// Mitsubishi GX Works2 project: yudomotmutistep   PLC: Q03UDV

PROGRAM MAIN
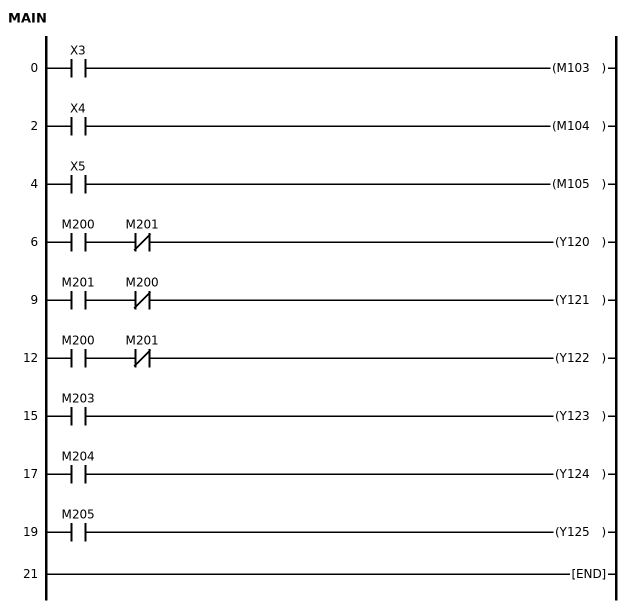
0     LD      X3
      OUT     M103
2     LD      X4
      OUT     M104
4     LD      X5
      OUT     M105
6     LD      M200
      ANI     M201
      OUT     Y120
9     LD      M201
      ANI     M200
      OUT     Y121
12    LD      M200
      ANI     M201
      OUT     Y122
15    LD      M203
      OUT     Y123
17    LD      M204
      OUT     Y124
19    LD      M205
      OUT     Y125
21    END
END_PROGRAM
